// This function has been automatically generated from the project information.
VAR_GLOBAL CONSTANT
	{attribute 'const_non_replaced'}
	stLibVersion_IO_DigiIn_Lib : ST_LibVersion := (iMajor := 1, iMinor := 0, iBuild := 0, iRevision := 0, sVersion := '1.0');
END_VAR

(* stored: Version 1.1.0.1, ProductVersion 3.1.0.36
   GVL Global_Version: Id {40fded1e-fb82-405a-931f-7e9c64d18290} *)
